PROGRAM MAIN
VAR
END_VAR

P_EnumeratorExample();
P_AdapterExample();
P_StringBuilderExample();

END_PROGRAM

(* stored: Version 1.1.0.1, ProductVersion 3.1.4024.4
   POU MAIN: Id {bb76c191-1e39-4156-925e-1a5af04519cc}, SpecialFunc None *)
